FUNCTION_BLOCK SizeMeasure
VAR_INPUT
END_VAR
VAR_OUTPUT
	//0-115cm
	sizeInCm : REAL;
END_VAR
VAR
	//0%-100%
	sizeInPercent : REAL;

    rawMin   : INT := 0;
    rawMax   : INT := 32767;
    scaledMin : REAL := 0.0;
    scaledMax : REAL := 115.0;
END_VAR

//Scaling
sizeInPercent := (scaledMax - scaledMin) / (rawMax - rawMin);
sizeInCm := scaledMin + (sizeInPercent * (inputs.Size_measure - rawMin));

END_FUNCTION_BLOCK

(* stored: Version 1.1.0.1, ProductVersion 3.1.4024.13
   POU SizeMeasure: Id {98e665cf-0e09-4803-b3b9-f218d0a86c5c}, SpecialFunc None *)
